Yaskawa INFORM job: SYS_SPINDLE_START.JBI

/JOB
//NAME SYS_SPINDLE_START
//POS
///NPOS 0,0,0,0,0,0
//INST
///DATE 2022/05/18 14:00
///ATTR SC,RW
///GROUP1 RB1
NOP
DOUT OT#(1) OFF
DOUT OT#(17) ON
WAIT T=1.00
DOUT OT#(1) ON
END
